{attribute 'qualified_only'}
VAR_GLOBAL
	rDist1 : LREAL; // distance in mm
END_VAR

(* stored: Version 1.1.0.1, ProductVersion 3.1.4024.11
   GVL GVL_HMI: Id {92c52021-3690-4c12-9801-36464fd60164} *)
